FUNCTION_BLOCK EL3021
VAR
	_io : EL3xx1_Data;
	{attribute addProperty Name "WcState"}
	_wcState : WcStateInputToggle;
	{attribute addProperty Name "Info data"}
	_infoData : InfoDataAds;
END_VAR

PROPERTY IO : REFERENCE TO EL3xx1_Data
GET
IO REF= _io;
END_GET
END_PROPERTY

PROPERTY WcState : REFERENCE TO WcStateInputToggle
GET
WcState REF= _wcState;
END_GET
END_PROPERTY

END_FUNCTION_BLOCK

(* stored: Version 1.1.0.1, ProductVersion 3.1.4024.9
   POU EL3021: Id {9a9cb86c-706b-0b70-024a-6e72f3ef76ed}, SpecialFunc None
   Property IO: Id {79b7a0ca-48c2-027b-2910-1493b0117d73}
   Get Get: Id {377b4de3-027c-08bf-2936-ea0a447c9380}
   Property WcState: Id {3bed4d84-26fb-0b9b-0f23-ffd10a8bce0a}
   Get Get: Id {105a46c7-cec2-0069-2b05-f8b3801440db} *)
